PROGRAM DistStationSensors
VAR
	StackLimit: WORD := 8; (* Stating the limit of the stack module barrel*)
	null: BOOL; (* set when stack module barrel is empty*)
	Current: WORD ; (* Current number of base/s in the stack module barrel*)
	LimitReached: BOOL; (* set when the stack module barrel is full*)
	counter1: CTUD;  (* counter used to count the number of bases inserted in the barrel*)
	
END_VAR
VAR // added by the converter: edge detectors and wires of the graphical bodies
    _w1, _w2, _w3, _w4 : BOOL;
END_VAR

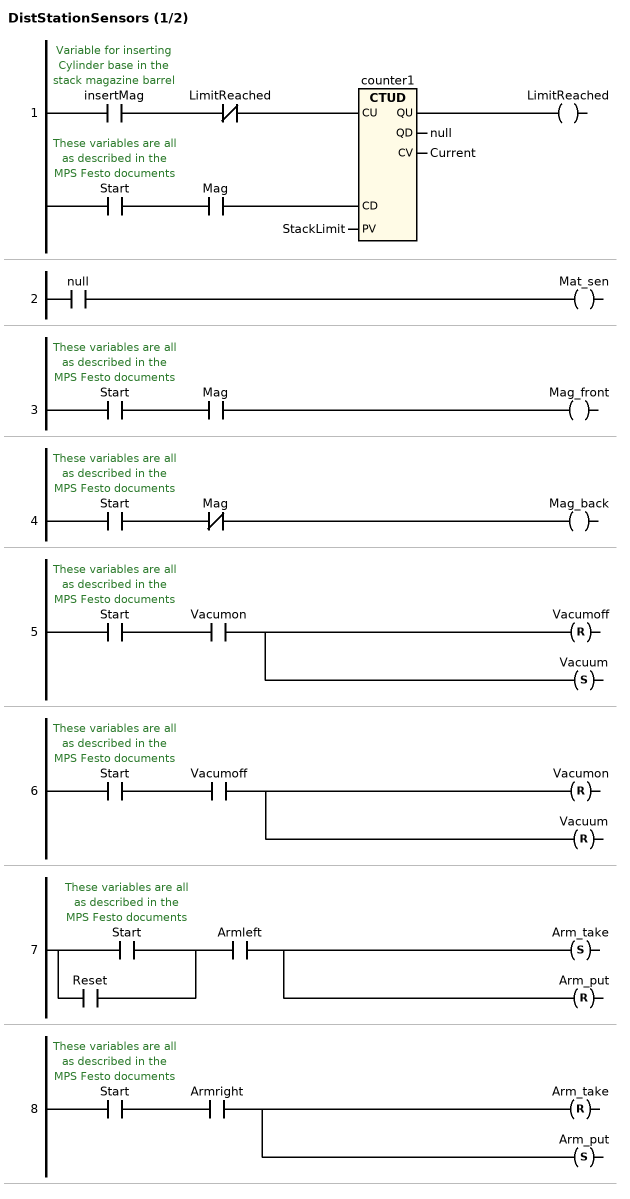
// NETWORK 1
//   insertMag: Variable for inserting Cylinder base in the stack magazine barrel
//   Start: These variables are all as described in the MPS Festo documents
counter1(
    CU := insertMag AND NOT LimitReached,
    CD := Start AND Mag,
    PV := StackLimit,
    QD => null,
    CV => Current); // CTUD
LimitReached := counter1.QU;

// NETWORK 2
Mat_sen := null;

// NETWORK 3
//   Start: These variables are all as described in the MPS Festo documents
Mag_front := Start AND Mag;

// NETWORK 4
//   Start: These variables are all as described in the MPS Festo documents
Mag_back := Start AND NOT Mag;

// NETWORK 5
//   Start: These variables are all as described in the MPS Festo documents
_w1 := Start AND Vacumon;
Vacumoff R= _w1;
Vacuum S= _w1;

// NETWORK 6
//   Start: These variables are all as described in the MPS Festo documents
_w2 := Start AND Vacumoff;
Vacumon R= _w2;
Vacuum R= _w2;

// NETWORK 7
//   Start: These variables are all as described in the MPS Festo documents
_w3 := (Start OR Reset) AND Armleft;
Arm_take S= _w3;
Arm_put R= _w3;

// NETWORK 8
//   Start: These variables are all as described in the MPS Festo documents
_w4 := Start AND Armright;
Arm_take R= _w4;
Arm_put S= _w4;

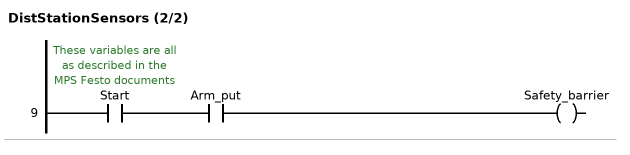
// NETWORK 9
//   Start: These variables are all as described in the MPS Festo documents
Safety_barrier := Start AND Arm_put;

END_PROGRAM

(* stored: Version 1.1.0.1, ProductVersion 3.1.4018.5
   POU DistStationSensors: Id {63acbffb-fc75-4cbe-934c-b62139645a0a}, SpecialFunc None *)
